// TIA Portal V20 export
ORGANIZATION_BLOCK "Main"   // OB123, LAD, ProgramCycle
TITLE = "Main Program Sweep (Cycle)"
// stored: Namespace ELY_1, SetENOAutomatically false
   VAR_INPUT
      Initial_Call : Bool;   // Initial call of this OB
      Remanence : Bool;   // =True, if remanent data are available
   END_VAR
BEGIN

REGION Network 1
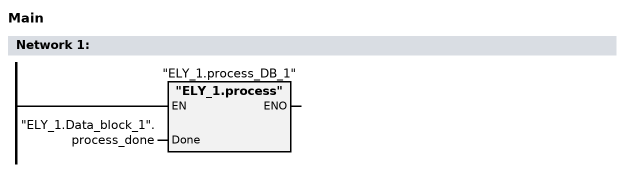
   RUNG wire#powerrail
      "ELY_1.process_DB_1"(Done := "ELY_1.Data_block_1".process_done)
   END_RUNG
   // the same network as SCL:
   "ELY_1.process_DB_1"(Done := "ELY_1.Data_block_1".process_done);   // "ELY_1.process"
END_REGION
END_ORGANIZATION_BLOCK
